PROGRAM main
VAR
	Start AT %QX0.0 : bool;
	StopPressed AT %QX0.1 : bool;
	SystemActive AT %QX0.2 : bool;
END_VAR

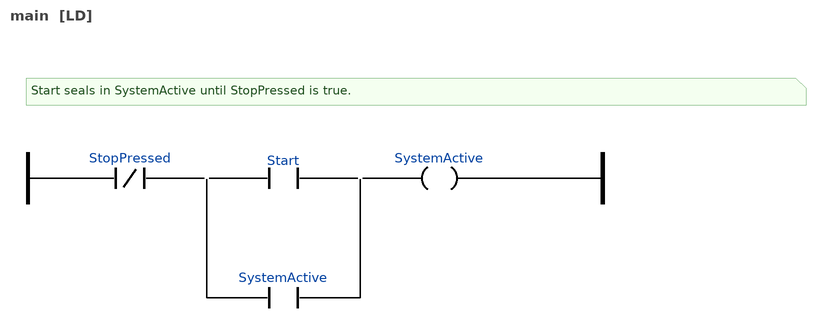
(* LD diagram, written out as Structured Text *)
(* Start seals in SystemActive until StopPressed is true. *)
SystemActive := NOT StopPressed AND (Start OR SystemActive);
END_PROGRAM
